FUNCTION_BLOCK AccumDDHHMM
VAR_INPUT
	State:BOOL;
	Retentive:BOOL;
	Reset:BOOL;
END_VAR

VAR PERSISTENT
	Mins:WORD;
	Hrs:WORD;
	Sec:WORD;
	Days:WORD;
END_VAR

VAR
	DispayTime:STRING;
	timer:TON;
	timerPT:TIME:=T#1M;
	StateToOff: F_TRIG;
    
END_VAR

VAR_TEMP
	displayTimeFormat: FB_FormatString;	
	foo:DINT;
END_VAR
VAR // added by the converter: edge detectors and wires of the graphical bodies
    _w1, _w2, _w3 : BOOL;
END_VAR

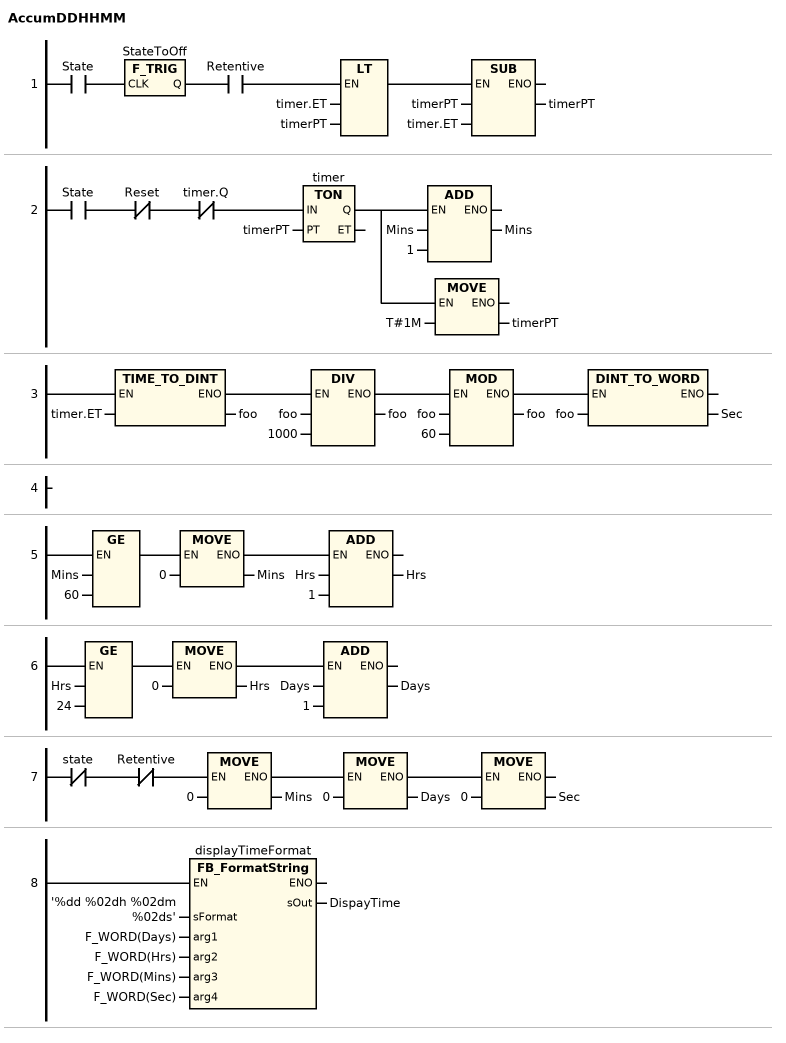
// NETWORK 1
StateToOff(CLK := State); // F_TRIG
IF StateToOff.Q AND Retentive AND timer.ET < timerPT THEN timerPT := timerPT - timer.ET; END_IF

// NETWORK 2
timer(IN := State AND NOT Reset AND NOT timer.Q, PT := timerPT); // TON
IF timer.Q THEN Mins := Mins + 1; END_IF
IF timer.Q THEN timerPT := T#1M; END_IF

// NETWORK 3
foo := TIME_TO_DINT(timer.ET);
foo := foo / 1000;
foo := foo MOD 60;
Sec := DINT_TO_WORD(foo);

// NETWORK 4

// NETWORK 5
_w1 := Mins >= 60;
IF _w1 THEN Mins := 0; END_IF
IF _w1 THEN Hrs := Hrs + 1; END_IF

// NETWORK 6
_w2 := Hrs >= 24;
IF _w2 THEN Hrs := 0; END_IF
IF _w2 THEN Days := Days + 1; END_IF

// NETWORK 7
_w3 := NOT state AND NOT Retentive;
IF _w3 THEN Mins := 0; END_IF
IF _w3 THEN Days := 0; END_IF
IF _w3 THEN Sec := 0; END_IF

// NETWORK 8
displayTimeFormat(
    sFormat := '%dd %02dh %02dm %02ds',
    arg1 := F_WORD(Days),
    arg2 := F_WORD(Hrs),
    arg3 := F_WORD(Mins),
    arg4 := F_WORD(Sec),
    sOut => DispayTime); // FB_FormatString

END_FUNCTION_BLOCK

(* stored: Version 1.1.0.1, ProductVersion 3.1.4024.12
   POU AccumDDHHMM: Id {409d937e-b3af-4cc1-9566-e4f7fac8e5cc}, SpecialFunc None *)
